PROGRAM MAIN
VAR
	// print out 'Hello world'
	fbStringBuilder : FB_StringBuilder;
	iStringBuilder	: I_StringBuilder := fbStringBuilder;
	sResult1 : STRING;
	sResult2 : STRING;
	bTest : BOOL;
END_VAR

IF bTest THEN
	// Function Block Instance
	sResult1 := fbStringBuilder.Clear()
							.Append('H')
							.Append('e')
							.Append('l')
							.Append('l')
							.Append('o')
							.Append(' ')
							.Append('W')
							.Append('o')
							.Append('r')
							.Append('l')
							.Append('d')
							.ToString();
	// Interface 
	sResult2 := iStringBuilder.Clear()
							.Append('H')
							.Append('e')
							.Append('l')
							.Append('l')
							.Append('o')
							.Append(' ')
							.Append('W')
							.Append('o')
							.Append('r')
							.Append('l')
							.Append('d')
							.ToString();
	bTest := FALSE;
END_IF

END_PROGRAM

(* stored: Version 1.1.0.1, ProductVersion 3.1.4024.12
   POU MAIN: Id {08544fae-b1ad-4dfc-82b7-0ab7f6e9ce50}, SpecialFunc None *)
